(*
  MAIN — Voorbeeld pompdrukregeling met FB_PompDrukPID
  =====================================================

  Aansluitschema:
    - Druksensor  : analoge ingang  (bv. 4-20mA of 0-10V -> geschaald naar bar)
    - Pompuitgang : analoge uitgang (0-100% -> bv. 0-10V naar frequentieregelaar)

  Uitgang minimum gedrag:
    - PID uitgang < rPompMin  => uitgang = 0.0  (pomp volledig UIT)
    - PID uitgang >= rPompMin => uitgang = berekende waarde (min. rPompMin)
    - PID uitgang > rPompMax  => uitgang = rPompMax
    Dit voorkomt dat de pomp op minimum blijft draaien als de druk al hoog genoeg is.

  Afstellen (aanbevolen volgorde):
    1. Start met Kp = 1.0, Ti = 0 (I uit), Td = 0
    2. Verhoog Kp tot lichte oscillatie, halveer dan Kp
    3. Voeg integratietijd Ti toe (begin bij 5-10s, verlaag tot gewenste nauwkeurigheid)
    4. Stel rSpRamp in als setpointsprongen een P-piek geven (bv. 0.5 bar/s)
    5. D is voor pompdruk normaal NIET nodig — laat Td = 0.0
*)
PROGRAM MAIN
VAR
    fbPompPID       : FB_PompDrukPID;

    // --- Proceswaarden ---
    rDrukSetpoint   : REAL := 3.0;   // Gewenste druk [bar]  — via HMI aanpasbaar
    rDrukMeting     : REAL;          // Gemeten druk [bar]   — van sensor

    // --- PID parameters (via HMI of variabelenlijst instelbaar) ---
    rKp             : REAL := 5.0;   // Proportionele versterking
    rTi             : REAL := 2.0;   // Integratietijd [s]  (0 = I uit)
    rTd             : REAL := 0.0;   // Differentiatietijd [s] (0 = D uit — aanbevolen)
    rSpRamp         : REAL := 0.5;   // Max setpointwijziging [bar/s] (0 = ramp uit)

    // --- Uitgang begrenzing ---
    rPompMin        : REAL := 20.0;  // Minimum loopsnelheid pomp [%]  (bij PID < min => 0%)
    rPompMax        : REAL := 100.0; // Maximum pompuitgang [%]
    rHysterese      : REAL := 5.0;   // Hysterese boven rPompMin voor inschakelen [%]
    rDoodband       : REAL := 0.2;   // Doodband rondom setpoint [bar] (0 = uit)
                                     // Geen P/I actie binnen ±0.2 bar van setpoint
    rMinAanTijd     : REAL := 5.0;   // Minimale aanlooptijd na elke start [s]
                                     // Pomp blijft min 5s aan na start (voorkomt direct uitschakelen)
    rMinLooptijd    : REAL := 30.0;  // Max tijd op minimum draaien [s] (0 = uit)
                                     // Na 30s op min => pomp uit, herstart bij druk < SP-doodband

    // --- Bediening ---
    bPIDActief      : BOOL := FALSE; // PID starten/stoppen
    bReset          : BOOL;          // Bumpless reset naar 0

    // --- Uitgang naar aandrijving ---
    rPompUitgang    : REAL;          // 0.0 of rPompMin..rPompMax [%]
END_VAR


// ---------------------------------------------------------------
// Druksensor inlezen — pas schalingsfactor aan op uw sensor
// Voorbeeld: 0-10V analoge ingang = 0-10 bar
//   rDrukMeting := GVL.rAI_DrukSensor * 10.0;
//
// Voorbeeld: 4-20mA = 0-16 bar (via 0-10V ingang via 500Ω shunt):
//   rDrukMeting := (GVL.rAI_DrukSensor - 2.0) / 8.0 * 16.0;
// ---------------------------------------------------------------

// PID aanroepen
fbPompPID(
    bEnable        := bPIDActief,
    rSetpoint      := rDrukSetpoint,
    rMeting        := rDrukMeting,
    rKp            := rKp,
    rTi            := rTi,
    rTd            := rTd,
    rSpRamp        := rSpRamp,
    rDoodband      := rDoodband,
    rUitMin        := rPompMin,
    rUitMax        := rPompMax,
    rHysterese     := rHysterese,
    rMinAanTijd    := rMinAanTijd,
    rMinLooptijd   := rMinLooptijd,
    rCyclustijd    := 0.01,          // Pas aan op uw task-periode (hier 10ms)
    bReset         := bReset
);

// Uitgang overnemen
// fbPompPID.rUitgang = 0.0 als PID < rPompMin, anders rPompMin..rPompMax
rPompUitgang := fbPompPID.rUitgang;

// ---------------------------------------------------------------
// Uitgang naar frequentieregelaar / pomp sturen
// Voorbeeld: 0-100% -> 0-10V analoge uitgang
//   GVL.rAO_PompSnelheid := rPompUitgang / 100.0 * 10.0;
// ---------------------------------------------------------------

END_PROGRAM

(* stored: Version 1.1.0.1, ProductVersion 3.1.4024.0
   POU MAIN: Id {b2c3d4e5-f6a7-8901-bcde-f12345678901}, SpecialFunc None *)
